# EPICS alarm handler configuration: mps_database/bare/alarms/areas/mpln_fees_mp01.alhConfig
GROUP NULL MPLN:FEES:MP01:1
$ALIAS MPS Link Node 216
$GUIDANCE
LTUH MPS
   Group Name: MPLN:FEES:MP01:1
   Summary PV:  MPLN:FEES:MP01:1:STATSUMY
$END
CHANNEL  MPLN:FEES:MP01:1    MPLN:FEES:MP01:1:MPS_EN_RBV		-----
CHANNEL  MPLN:FEES:MP01:1    MPLN:FEES:MP01:1:LC1_MODE_RBV		-----
